// TIA Portal project "Project-Sticle" (V15.1)

(* hardware
DEVICE "S71500/ET200MP station_1"  S7-1500 station
   slot 0: "Rail_0"  Rack  6ES7 590-1***0-0AA0
   slot 1: "PLC_1"  CPU 1513-1 PN  6ES7 513-1AL02-0AB0  V2.6
      slot 3: "CPU display_1"  6ES7591-1AA00-0AA0
*)

// ===== PLC "PLC_1"  CPU 1513-1 PN =====

VAR_GLOBAL   // PLC tag table "Default tag table"
   "Clock_Byte" AT %MB0 : Byte;
   "Clock_10Hz" AT %M0.0 : Bool;
   "Clock_5Hz" AT %M0.1 : Bool;
   "Clock_2.5Hz" AT %M0.2 : Bool;
   "Clock_2Hz" AT %M0.3 : Bool;
   "Clock_1.25Hz" AT %M0.4 : Bool;
   "Clock_1Hz" AT %M0.5 : Bool;
   "Clock_0.625Hz" AT %M0.6 : Bool;
   "Clock_0.5Hz" AT %M0.7 : Bool;
END_VAR

DATA_BLOCK "Avarii"   // DB1
{ S7_Optimized_Access := 'TRUE' }
VERSION : 0.1
   VAR
      esd : Bool;
      esd_btn : Bool;
      reset_esd : Bool;
      confirmare_neprimita_actuator : Bool;
      reset_avarii : Bool;
      avarie_imbuteliere : Bool;
      avarie_capace : Bool;
      avarie_eticheta : Bool;
      avarie_impachetare : Bool;
      avarie_generala : Bool;
   END_VAR
BEGIN
END_DATA_BLOCK

DATA_BLOCK "Alarme"   // DB2
{ S7_Optimized_Access := 'TRUE' }
VERSION : 0.1
   VAR
      alarme_gather : Word;
      alarme_vect : Array[0..15] of Bool;
   END_VAR
BEGIN
END_DATA_BLOCK

DATA_BLOCK "Senzori"   // DB3
{ S7_Optimized_Access := 'TRUE' }
VERSION : 0.1
   VAR
      completat_1 : UInt;
   END_VAR
BEGIN
END_DATA_BLOCK

DATA_BLOCK "Banda"   // DB4
{ S7_Optimized_Access := 'TRUE' }
VERSION : 0.1
   VAR
      banda_pornita_1 : Bool;
      prm_pornire_banda11 : Bool;
      prm_pornire_banda12 : Bool;
      banda_oprita_2 : Bool;
      banda_oprita_3 : Bool;
      banda_oprita_4 : Bool;
   END_VAR
BEGIN
END_DATA_BLOCK

DATA_BLOCK "Aparate"   // DB5
{ S7_Optimized_Access := 'TRUE' }
VERSION : 0.1
   VAR
      numar_sticle_cerut : UInt;
      numar_sticle : UInt;
      inchidere_actuator : Bool;
      deschidere_actuator : Bool;
      confirmare_actuator : Bool;
      timp_umplere_user : Time;
      timp_umplere_secunde : Time;
      terminat_imbuteliere : Bool;
      ajuns_capace : Bool;
      plecat_capace : Bool;
      ajuns_eticheta : Bool;
      plecat_ethicheta : Bool;
      ajuns_impachetare : Bool;
      plecat_impachetare : Bool;
   END_VAR
BEGIN
END_DATA_BLOCK

DATA_BLOCK "Butoane/Permisiuni"   // DB6
{ S7_Optimized_Access := 'TRUE' }
VERSION : 0.1
   VAR
      btn_start : Bool;
      permisiune_start : Bool;
      nr_sticle_complet : Bool;
   END_VAR
BEGIN
END_DATA_BLOCK

DATA_BLOCK "Rising_edges"   // DB7
{ S7_Optimized_Access := 'TRUE' }
VERSION : 0.1
   VAR
      re1 : Bool;
      re2 : Bool;
      re3 : Bool;
   END_VAR
BEGIN
END_DATA_BLOCK

DATA_BLOCK "Hysteresis_DB"   // DB15
{ S7_Optimized_Access := 'TRUE' }
VERSION : 0.1
// stored: InstanceOfName Hysteresis
"Hysteresis"
BEGIN
END_DATA_BLOCK

DATA_BLOCK "Variabile_Hysteresis"   // DB16
{ S7_Optimized_Access := 'TRUE' }
VERSION : 0.1
   VAR
      bool_cond : Bool;
      Hy_val : Real;
      Setpoint : Real;
      temp : Real;
      lim_inf : Real;
      lim_sup : Real;
   END_VAR
BEGIN
END_DATA_BLOCK

// folder: System blocks/Program resources

DATA_BLOCK "timer_confirmare_actuator"   // DB8
{ S7_Optimized_Access := 'TRUE' }
AUTHOR : Simatic
FAMILY : IEC
NAME : IEC_TMR
VERSION : 1.0
// stored: InstanceOfName IEC_TIMER
"IEC_TIMER"
BEGIN
END_DATA_BLOCK

DATA_BLOCK "timer_imbuteliere"   // DB9
{ S7_Optimized_Access := 'TRUE' }
AUTHOR : Simatic
FAMILY : IEC
NAME : IEC_TMR
VERSION : 1.0
// stored: InstanceOfName IEC_TIMER
"IEC_TIMER"
BEGIN
END_DATA_BLOCK

DATA_BLOCK "timer_reset_btn_avarii"   // DB10
{ S7_Optimized_Access := 'TRUE' }
AUTHOR : Simatic
FAMILY : IEC
NAME : IEC_TMR
VERSION : 1.0
// stored: InstanceOfName IEC_TIMER
"IEC_TIMER"
BEGIN
END_DATA_BLOCK

DATA_BLOCK "timer_capace"   // DB11
{ S7_Optimized_Access := 'TRUE' }
AUTHOR : Simatic
FAMILY : IEC
NAME : IEC_TMR
VERSION : 1.0
// stored: InstanceOfName IEC_TIMER
"IEC_TIMER"
BEGIN
END_DATA_BLOCK

DATA_BLOCK "timer_eticheta"   // DB12
{ S7_Optimized_Access := 'TRUE' }
AUTHOR : Simatic
FAMILY : IEC
NAME : IEC_TMR
VERSION : 1.0
// stored: InstanceOfName IEC_TIMER
"IEC_TIMER"
BEGIN
END_DATA_BLOCK

DATA_BLOCK "timer_impachetare"   // DB13
{ S7_Optimized_Access := 'TRUE' }
AUTHOR : Simatic
FAMILY : IEC
NAME : IEC_TMR
VERSION : 1.0
// stored: InstanceOfName IEC_TIMER
"IEC_TIMER"
BEGIN
END_DATA_BLOCK

DATA_BLOCK "reset_esd"   // DB14
{ S7_Optimized_Access := 'TRUE' }
AUTHOR : Simatic
FAMILY : IEC
NAME : IEC_TMR
VERSION : 1.0
// stored: InstanceOfName IEC_TIMER
"IEC_TIMER"
BEGIN
END_DATA_BLOCK

// folder: (top level)

FUNCTION_BLOCK "Hysteresis"   // FB1, LAD
{ S7_Optimized_Access := 'TRUE' }
VERSION : 0.1
   VAR_INPUT
      HY_val : Real;
      Setpoint : Real;
   END_VAR
   VAR_OUTPUT
      h_lim_sup : Real;
      h_lim_inf : Real;
      bool_cond : Bool;
   END_VAR
   VAR_IN_OUT
      temp : Real;
   END_VAR
   VAR
      re1 : Bool;
      re2 : Bool;
      urcare : Bool;
   END_VAR
   VAR_TEMP   // added for the SCL form of the ladder/FBD networks
      _w1 : Bool;
   END_VAR
BEGIN

REGION Network 1: daca are comanda de bool, sa creasca
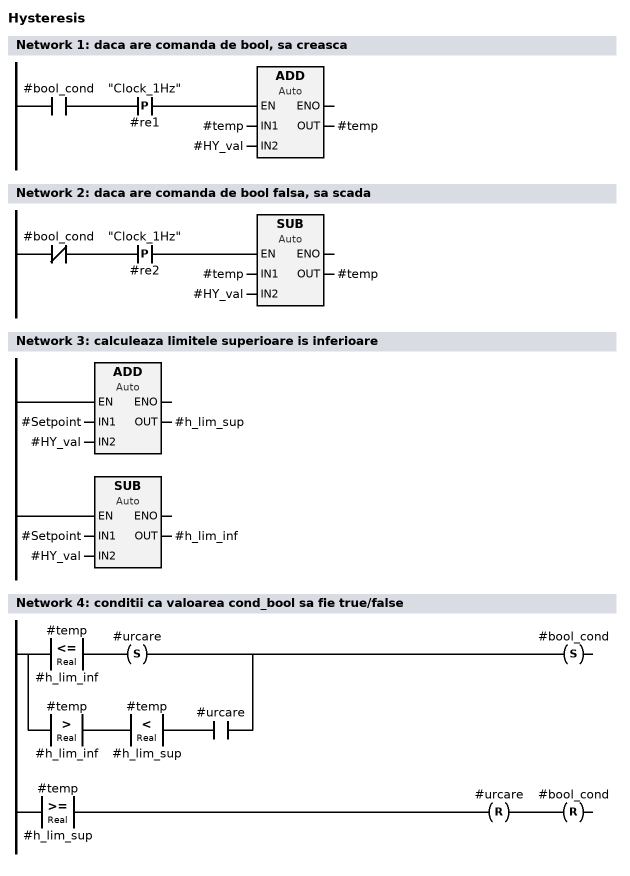
   RUNG wire#powerrail
      Contact( #bool_cond )
      P_Contact(operand := "Clock_1Hz", bit := #re1)
      Add(in1 := #temp, in2 := #HY_val, out => #temp)
   END_RUNG
   // the same network as SCL:
   #_w1 := #bool_cond AND "Clock_1Hz" AND NOT #re1;   // rising edge of "Clock_1Hz"
   #re1 := "Clock_1Hz";
   IF #_w1 THEN #temp := #temp + #HY_val; END_IF;
END_REGION

REGION Network 2: daca are comanda de bool falsa, sa scada
   RUNG wire#powerrail
      I_Contact( #bool_cond )
      P_Contact(operand := "Clock_1Hz", bit := #re2)
      Sub(in1 := #temp, in2 := #HY_val, out => #temp)
   END_RUNG
   // the same network as SCL:
   #_w1 := NOT #bool_cond AND "Clock_1Hz" AND NOT #re2;   // rising edge of "Clock_1Hz"
   #re2 := "Clock_1Hz";
   IF #_w1 THEN #temp := #temp - #HY_val; END_IF;
END_REGION

REGION Network 3: calculeaza limitele superioare is inferioare
   RUNG wire#powerrail
      Add(in1 := #Setpoint, in2 := #HY_val, out => #h_lim_sup)
   END_RUNG
   RUNG wire#powerrail
      Sub(in1 := #Setpoint, in2 := #HY_val, out => #h_lim_inf)
   END_RUNG
   // the same network as SCL:
   #h_lim_sup := #Setpoint + #HY_val;
   #h_lim_inf := #Setpoint - #HY_val;
END_REGION

REGION Network 4: conditii ca valoarea cond_bool sa fie true/false
   RUNG wire#powerrail
      { S7_Templates := "SrcType := Real" } LE_Contact(in1 := #temp, in2 := #h_lim_inf)
      S_Coil( #urcare )
      wire#w1
      S_Coil( #bool_cond )
   END_RUNG
   RUNG wire#powerrail
      { S7_Templates := "SrcType := Real" } GT_Contact(in1 := #temp, in2 := #h_lim_inf)
      { S7_Templates := "SrcType := Real" } LT_Contact(in1 := #temp, in2 := #h_lim_sup)
      Contact( #urcare )
   END_RUNG wire#w1
   RUNG wire#powerrail
      { S7_Templates := "SrcType := Real" } GE_Contact(in1 := #temp, in2 := #h_lim_sup)
      R_Coil( #urcare )
      R_Coil( #bool_cond )
   END_RUNG
   // the same network as SCL:
   #_w1 := #temp <= #h_lim_inf;
   IF #_w1 THEN #urcare := TRUE; END_IF;
   IF #_w1 OR ((#temp > #h_lim_inf) AND (#temp < #h_lim_sup) AND #urcare) THEN #bool_cond := TRUE; END_IF;
   IF #temp >= #h_lim_sup THEN
       #urcare := FALSE;
       #bool_cond := FALSE;
   END_IF;
END_REGION
END_FUNCTION_BLOCK

ORGANIZATION_BLOCK "Main"   // OB1, LAD, ProgramCycle
TITLE = "Main Program Sweep (Cycle)"
{ S7_Optimized_Access := 'TRUE' }
VERSION : 0.1
   VAR_INPUT
      Initial_Call : Bool;   // Initial call of this OB
      Remanence : Bool;   // =True, if remanent data are available
   END_VAR
   VAR_TEMP   // added for the SCL form of the ladder/FBD networks
      _w1 : Bool;
   END_VAR
BEGIN

REGION Network 1: permisiune start(adauga la final si avarie generala pt fiecare aparat in parte)
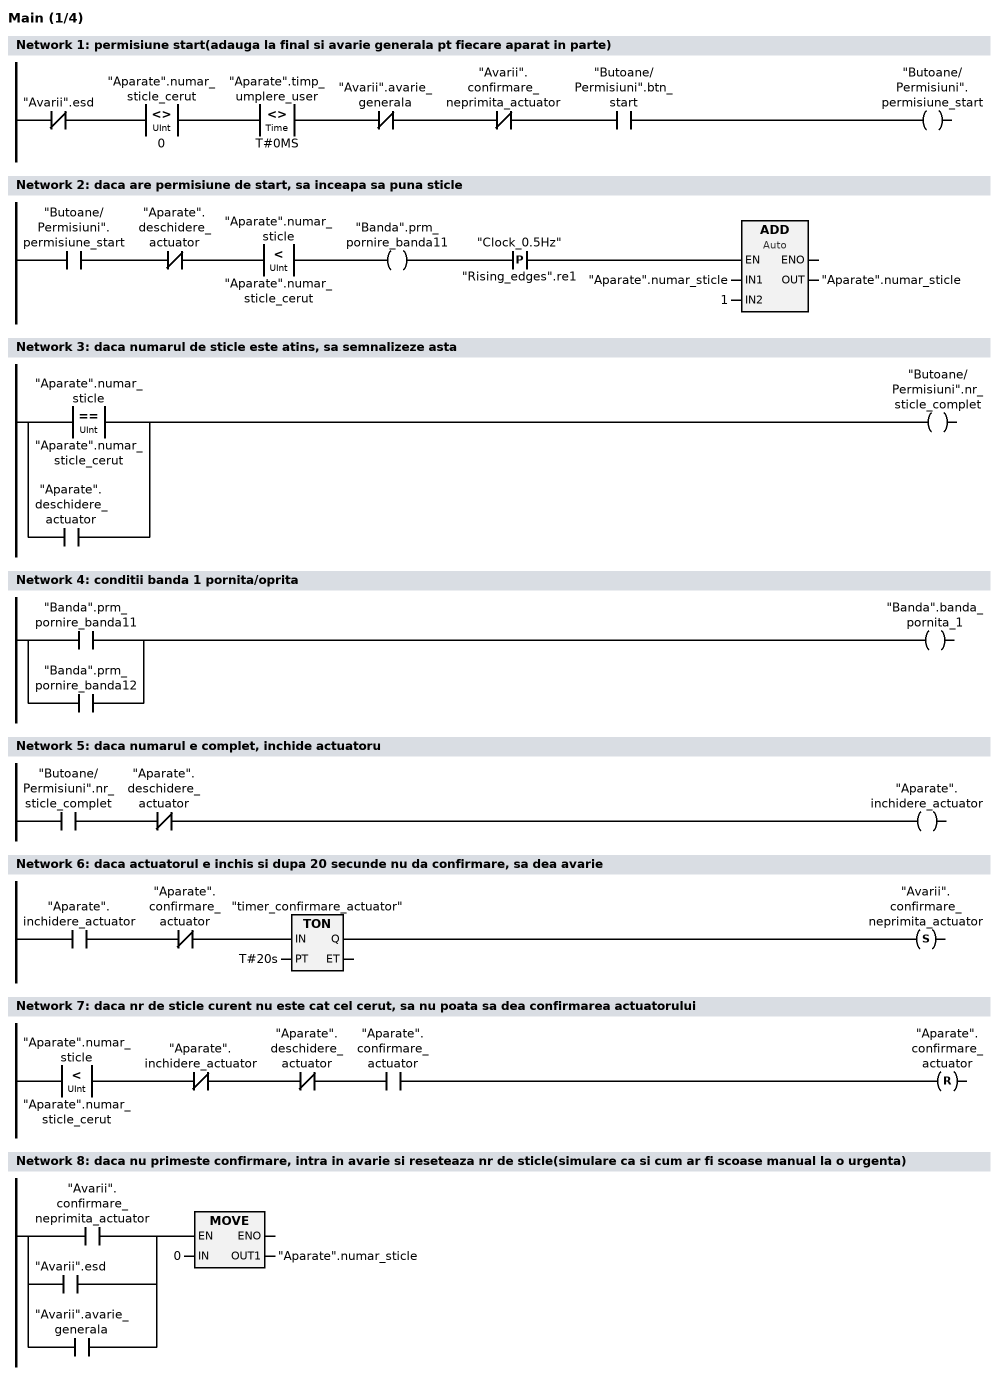
   RUNG wire#powerrail
      I_Contact( "Avarii".esd )
      { S7_Templates := "SrcType := UInt" } NE_Contact(in1 := "Aparate".numar_sticle_cerut, in2 := 0)
      { S7_Templates := "SrcType := Time" } NE_Contact(in1 := "Aparate".timp_umplere_user, in2 := T#0MS)
      I_Contact( "Avarii".avarie_generala )
      I_Contact( "Avarii".confirmare_neprimita_actuator )
      Contact( "Butoane/Permisiuni".btn_start )
      Coil( "Butoane/Permisiuni".permisiune_start )
   END_RUNG
   // the same network as SCL:
   "Butoane/Permisiuni".permisiune_start := NOT "Avarii".esd AND ("Aparate".numar_sticle_cerut <> 0) AND ("Aparate".timp_umplere_user <> T#0MS) AND NOT "Avarii".avarie_generala AND NOT "Avarii".confirmare_neprimita_actuator AND "Butoane/Permisiuni".btn_start;
END_REGION

REGION Network 2: daca are permisiune de start, sa inceapa sa puna sticle
   RUNG wire#powerrail
      Contact( "Butoane/Permisiuni".permisiune_start )
      I_Contact( "Aparate".deschidere_actuator )
      { S7_Templates := "SrcType := UInt" } LT_Contact(in1 := "Aparate".numar_sticle, in2 := "Aparate".numar_sticle_cerut)
      Coil( "Banda".prm_pornire_banda11 )
      P_Contact(operand := "Clock_0.5Hz", bit := "Rising_edges".re1)
      Add(in1 := "Aparate".numar_sticle, in2 := 1, out => "Aparate".numar_sticle)
   END_RUNG
   // the same network as SCL:
   "Banda".prm_pornire_banda11 := "Butoane/Permisiuni".permisiune_start AND NOT "Aparate".deschidere_actuator AND ("Aparate".numar_sticle < "Aparate".numar_sticle_cerut);
   #_w1 := "Banda".prm_pornire_banda11 AND "Clock_0.5Hz" AND NOT "Rising_edges".re1;   // rising edge of "Clock_0.5Hz"
   "Rising_edges".re1 := "Clock_0.5Hz";
   IF #_w1 THEN "Aparate".numar_sticle := "Aparate".numar_sticle + 1; END_IF;
END_REGION

REGION Network 3: daca numarul de sticle este atins, sa semnalizeze asta
   RUNG wire#powerrail
      { S7_Templates := "SrcType := UInt" } EQ_Contact(in1 := "Aparate".numar_sticle, in2 := "Aparate".numar_sticle_cerut)
      wire#w1
      Coil( "Butoane/Permisiuni".nr_sticle_complet )
   END_RUNG
   RUNG wire#powerrail
      Contact( "Aparate".deschidere_actuator )
   END_RUNG wire#w1
   // the same network as SCL:
   "Butoane/Permisiuni".nr_sticle_complet := ("Aparate".numar_sticle = "Aparate".numar_sticle_cerut) OR "Aparate".deschidere_actuator;
END_REGION

REGION Network 4: conditii banda 1 pornita/oprita
   RUNG wire#powerrail
      Contact( "Banda".prm_pornire_banda11 )
      wire#w1
      Coil( "Banda".banda_pornita_1 )
   END_RUNG
   RUNG wire#powerrail
      Contact( "Banda".prm_pornire_banda12 )
   END_RUNG wire#w1
   // the same network as SCL:
   "Banda".banda_pornita_1 := "Banda".prm_pornire_banda11 OR "Banda".prm_pornire_banda12;
END_REGION

REGION Network 5: daca numarul e complet, inchide actuatoru
   RUNG wire#powerrail
      Contact( "Butoane/Permisiuni".nr_sticle_complet )
      I_Contact( "Aparate".deschidere_actuator )
      Coil( "Aparate".inchidere_actuator )
   END_RUNG
   // the same network as SCL:
   "Aparate".inchidere_actuator := "Butoane/Permisiuni".nr_sticle_complet AND NOT "Aparate".deschidere_actuator;
END_REGION

REGION Network 6: daca actuatorul e inchis si dupa 20 secunde nu da confirmare, sa dea avarie
   "timer_confirmare_actuator".TON(IN := "Aparate".inchidere_actuator AND NOT "Aparate".confirmare_actuator,
                           PT := T#20s);
   IF "timer_confirmare_actuator".Q THEN "Avarii".confirmare_neprimita_actuator := TRUE; END_IF;
END_REGION

REGION Network 7: daca nr de sticle curent nu este cat cel cerut, sa nu poata sa dea confirmarea actuatorului
   RUNG wire#powerrail
      { S7_Templates := "SrcType := UInt" } LT_Contact(in1 := "Aparate".numar_sticle, in2 := "Aparate".numar_sticle_cerut)
      I_Contact( "Aparate".inchidere_actuator )
      I_Contact( "Aparate".deschidere_actuator )
      Contact( "Aparate".confirmare_actuator )
      R_Coil( "Aparate".confirmare_actuator )
   END_RUNG
   // the same network as SCL:
   IF ("Aparate".numar_sticle < "Aparate".numar_sticle_cerut) AND NOT "Aparate".inchidere_actuator AND NOT "Aparate".deschidere_actuator AND "Aparate".confirmare_actuator THEN
       "Aparate".confirmare_actuator := FALSE;
   END_IF;
END_REGION

REGION Network 8: daca nu primeste confirmare, intra in avarie si reseteaza nr de sticle(simulare ca si cum ar fi scoase manual la o urgenta)
   RUNG wire#powerrail
      Contact( "Avarii".confirmare_neprimita_actuator )
      wire#w1
      Move(in := 0, out1 => "Aparate".numar_sticle)
   END_RUNG
   RUNG wire#powerrail
      Contact( "Avarii".esd )
   END_RUNG wire#w1
   RUNG wire#powerrail
      Contact( "Avarii".avarie_generala )
   END_RUNG wire#w1
   // the same network as SCL:
   IF "Avarii".confirmare_neprimita_actuator OR "Avarii".esd OR "Avarii".avarie_generala THEN
       "Aparate".numar_sticle := 0;
   END_IF;
END_REGION

REGION Network 9: timp in secunde de la user pt umplere
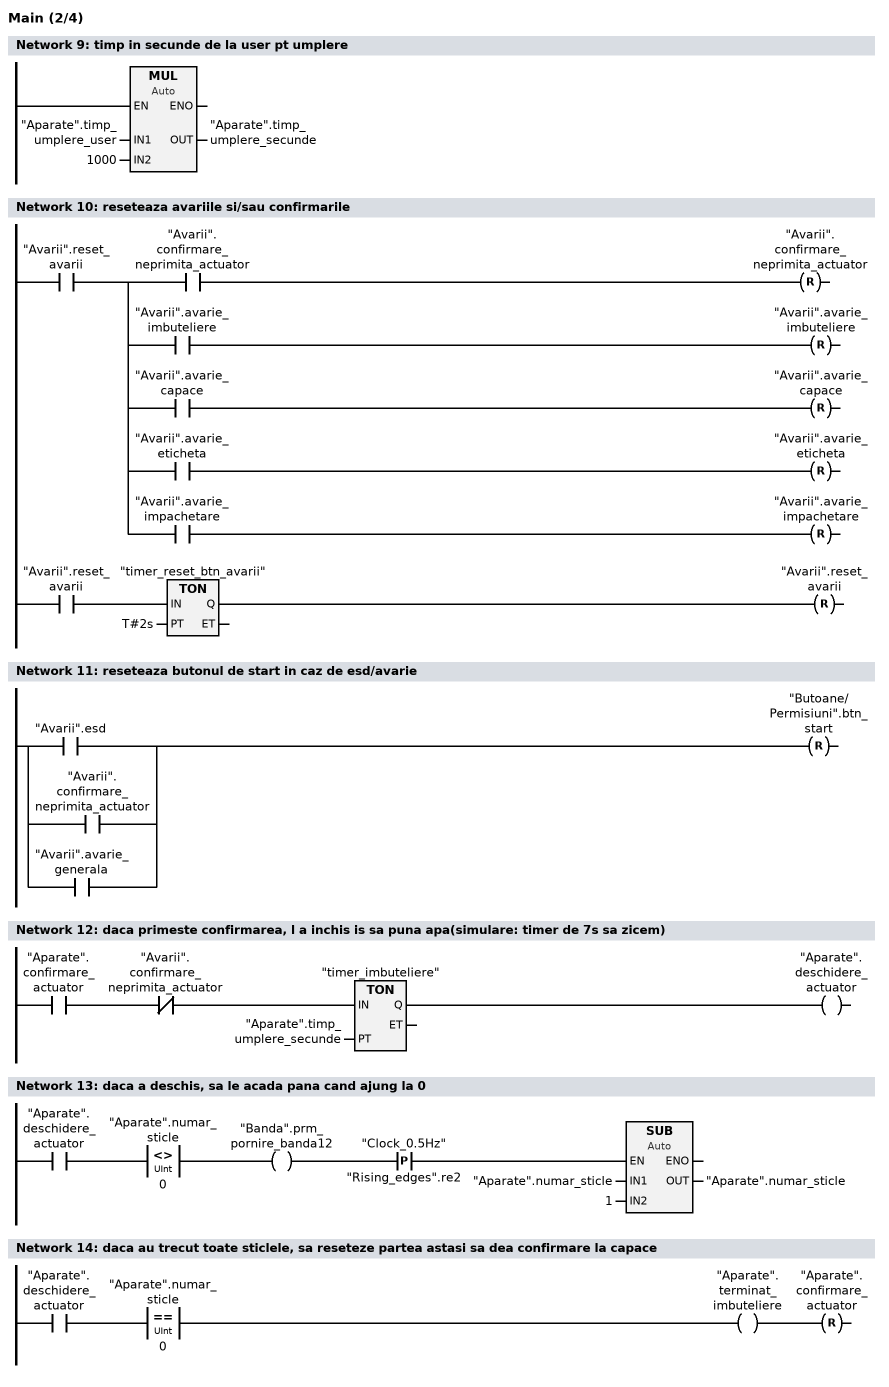
   RUNG wire#powerrail
      Mul(in1 := "Aparate".timp_umplere_user, in2 := 1000, out => "Aparate".timp_umplere_secunde)
   END_RUNG
   // the same network as SCL:
   "Aparate".timp_umplere_secunde := "Aparate".timp_umplere_user * 1000;
END_REGION

REGION Network 10: reseteaza avariile si/sau confirmarile
   IF "Avarii".reset_avarii AND "Avarii".confirmare_neprimita_actuator THEN
       "Avarii".confirmare_neprimita_actuator := FALSE;
   END_IF;
   IF "Avarii".reset_avarii AND "Avarii".avarie_imbuteliere THEN
       "Avarii".avarie_imbuteliere := FALSE;
   END_IF;
   IF "Avarii".reset_avarii AND "Avarii".avarie_capace THEN "Avarii".avarie_capace := FALSE; END_IF;
   IF "Avarii".reset_avarii AND "Avarii".avarie_eticheta THEN "Avarii".avarie_eticheta := FALSE; END_IF;
   IF "Avarii".reset_avarii AND "Avarii".avarie_impachetare THEN
       "Avarii".avarie_impachetare := FALSE;
   END_IF;
   "timer_reset_btn_avarii".TON(IN := "Avarii".reset_avarii, PT := T#2s);
   IF "timer_reset_btn_avarii".Q THEN "Avarii".reset_avarii := FALSE; END_IF;
END_REGION

REGION Network 11: reseteaza butonul de start in caz de esd/avarie
   RUNG wire#powerrail
      Contact( "Avarii".esd )
      wire#w1
      R_Coil( "Butoane/Permisiuni".btn_start )
   END_RUNG
   RUNG wire#powerrail
      Contact( "Avarii".confirmare_neprimita_actuator )
   END_RUNG wire#w1
   RUNG wire#powerrail
      Contact( "Avarii".avarie_generala )
   END_RUNG wire#w1
   // the same network as SCL:
   IF "Avarii".esd OR "Avarii".confirmare_neprimita_actuator OR "Avarii".avarie_generala THEN
       "Butoane/Permisiuni".btn_start := FALSE;
   END_IF;
END_REGION

REGION Network 12: daca primeste confirmarea, l a inchis is sa puna apa(simulare: timer de 7s sa zicem)
   "timer_imbuteliere".TON(IN := "Aparate".confirmare_actuator AND NOT "Avarii".confirmare_neprimita_actuator,
                           PT := "Aparate".timp_umplere_secunde);
   "Aparate".deschidere_actuator := "timer_imbuteliere".Q;
END_REGION

REGION Network 13: daca a deschis, sa le acada pana cand ajung la 0
   RUNG wire#powerrail
      Contact( "Aparate".deschidere_actuator )
      { S7_Templates := "SrcType := UInt" } NE_Contact(in1 := "Aparate".numar_sticle, in2 := 0)
      Coil( "Banda".prm_pornire_banda12 )
      P_Contact(operand := "Clock_0.5Hz", bit := "Rising_edges".re2)
      Sub(in1 := "Aparate".numar_sticle, in2 := 1, out => "Aparate".numar_sticle)
   END_RUNG
   // the same network as SCL:
   "Banda".prm_pornire_banda12 := "Aparate".deschidere_actuator AND ("Aparate".numar_sticle <> 0);
   #_w1 := "Banda".prm_pornire_banda12 AND "Clock_0.5Hz" AND NOT "Rising_edges".re2;   // rising edge of "Clock_0.5Hz"
   "Rising_edges".re2 := "Clock_0.5Hz";
   IF #_w1 THEN "Aparate".numar_sticle := "Aparate".numar_sticle - 1; END_IF;
END_REGION

REGION Network 14: daca au trecut toate sticlele, sa reseteze partea astasi sa dea confirmare la capace
   RUNG wire#powerrail
      Contact( "Aparate".deschidere_actuator )
      { S7_Templates := "SrcType := UInt" } EQ_Contact(in1 := "Aparate".numar_sticle, in2 := 0)
      Coil( "Aparate".terminat_imbuteliere )
      R_Coil( "Aparate".confirmare_actuator )
   END_RUNG
   // the same network as SCL:
   "Aparate".terminat_imbuteliere := "Aparate".deschidere_actuator AND ("Aparate".numar_sticle = 0);
   IF "Aparate".terminat_imbuteliere THEN "Aparate".confirmare_actuator := FALSE; END_IF;
END_REGION

REGION Network 15: daca a terminat imbutelierea, sa seteze ca a ajuns la capace
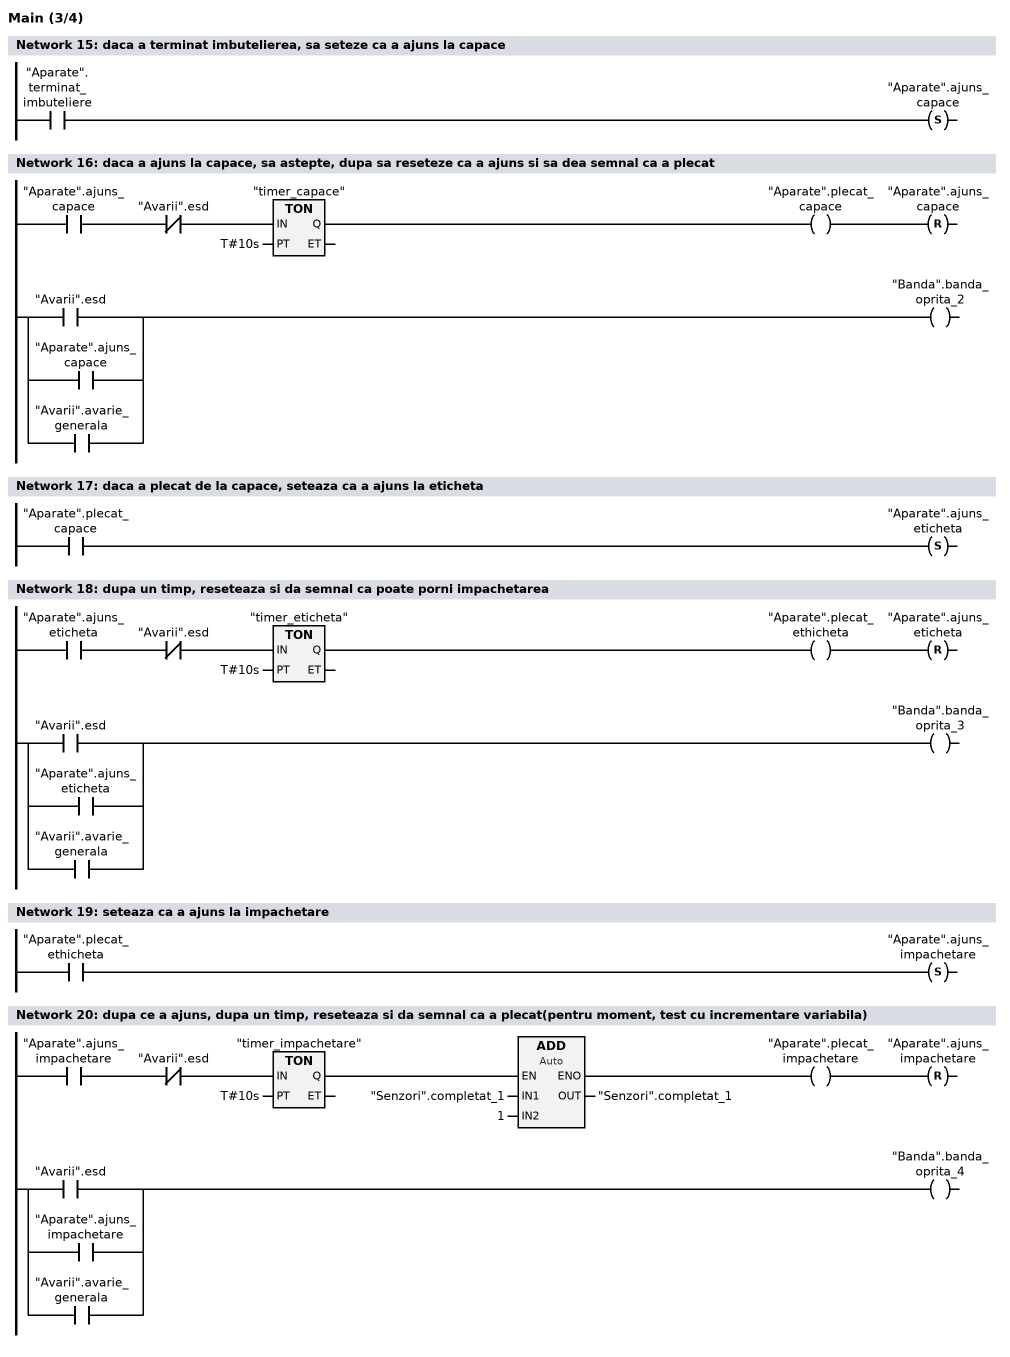
   RUNG wire#powerrail
      Contact( "Aparate".terminat_imbuteliere )
      S_Coil( "Aparate".ajuns_capace )
   END_RUNG
   // the same network as SCL:
   IF "Aparate".terminat_imbuteliere THEN "Aparate".ajuns_capace := TRUE; END_IF;
END_REGION

REGION Network 16: daca a ajuns la capace, sa astepte, dupa sa reseteze ca a ajuns si sa dea semnal ca a plecat
   "timer_capace".TON(IN := "Aparate".ajuns_capace AND NOT "Avarii".esd, PT := T#10s);
   "Aparate".plecat_capace := "timer_capace".Q;
   IF "timer_capace".Q THEN "Aparate".ajuns_capace := FALSE; END_IF;
   "Banda".banda_oprita_2 := "Avarii".esd OR "Aparate".ajuns_capace OR "Avarii".avarie_generala;
END_REGION

REGION Network 17: daca a plecat de la capace, seteaza ca a ajuns la eticheta
   RUNG wire#powerrail
      Contact( "Aparate".plecat_capace )
      S_Coil( "Aparate".ajuns_eticheta )
   END_RUNG
   // the same network as SCL:
   IF "Aparate".plecat_capace THEN "Aparate".ajuns_eticheta := TRUE; END_IF;
END_REGION

REGION Network 18: dupa un timp, reseteaza si da semnal ca poate porni impachetarea
   "timer_eticheta".TON(IN := "Aparate".ajuns_eticheta AND NOT "Avarii".esd, PT := T#10s);
   "Aparate".plecat_ethicheta := "timer_eticheta".Q;
   IF "timer_eticheta".Q THEN "Aparate".ajuns_eticheta := FALSE; END_IF;
   "Banda".banda_oprita_3 := "Avarii".esd OR "Aparate".ajuns_eticheta OR "Avarii".avarie_generala;
END_REGION

REGION Network 19: seteaza ca a ajuns la impachetare
   RUNG wire#powerrail
      Contact( "Aparate".plecat_ethicheta )
      S_Coil( "Aparate".ajuns_impachetare )
   END_RUNG
   // the same network as SCL:
   IF "Aparate".plecat_ethicheta THEN "Aparate".ajuns_impachetare := TRUE; END_IF;
END_REGION

REGION Network 20: dupa ce a ajuns, dupa un timp, reseteaza si da semnal ca a plecat(pentru moment, test cu incrementare variabila)
   "timer_impachetare".TON(IN := "Aparate".ajuns_impachetare AND NOT "Avarii".esd, PT := T#10s);
   IF "timer_impachetare".Q THEN "Senzori".completat_1 := "Senzori".completat_1 + 1; END_IF;
   "Aparate".plecat_impachetare := "timer_impachetare".Q;
   IF "timer_impachetare".Q THEN "Aparate".ajuns_impachetare := FALSE; END_IF;
   "Banda".banda_oprita_4 := "Avarii".esd OR "Aparate".ajuns_impachetare OR "Avarii".avarie_generala;
END_REGION

REGION Network 21: esd btn
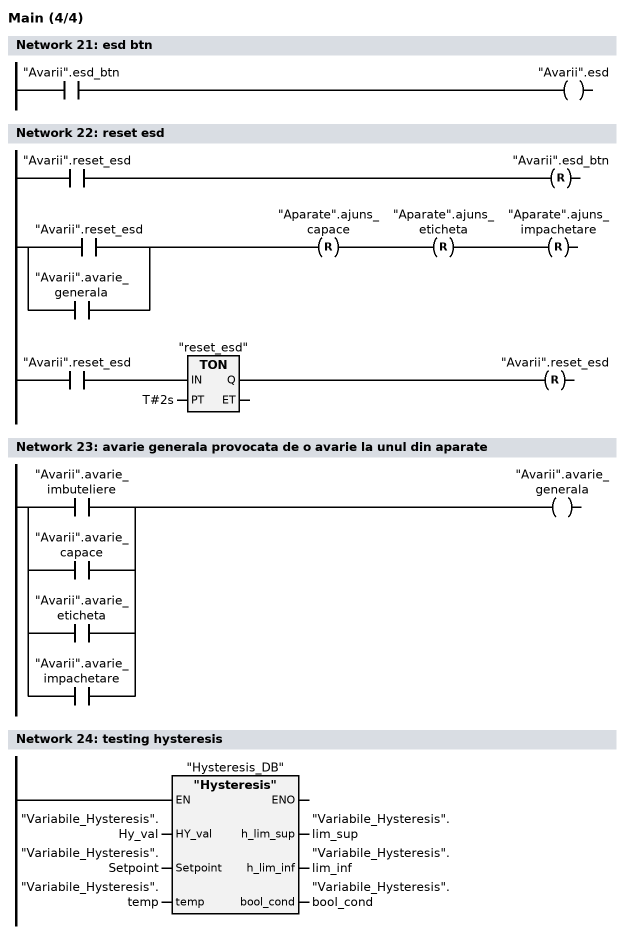
   RUNG wire#powerrail
      Contact( "Avarii".esd_btn )
      Coil( "Avarii".esd )
   END_RUNG
   // the same network as SCL:
   "Avarii".esd := "Avarii".esd_btn;
END_REGION

REGION Network 22: reset esd
   IF "Avarii".reset_esd THEN "Avarii".esd_btn := FALSE; END_IF;
   IF "Avarii".reset_esd OR "Avarii".avarie_generala THEN
       "Aparate".ajuns_capace := FALSE;
       "Aparate".ajuns_eticheta := FALSE;
       "Aparate".ajuns_impachetare := FALSE;
   END_IF;
   "reset_esd".TON(IN := "Avarii".reset_esd, PT := T#2s);
   IF "reset_esd".Q THEN "Avarii".reset_esd := FALSE; END_IF;
END_REGION

REGION Network 23: avarie generala provocata de o avarie la unul din aparate
   RUNG wire#powerrail
      Contact( "Avarii".avarie_imbuteliere )
      wire#w1
      Coil( "Avarii".avarie_generala )
   END_RUNG
   RUNG wire#powerrail
      Contact( "Avarii".avarie_capace )
   END_RUNG wire#w1
   RUNG wire#powerrail
      Contact( "Avarii".avarie_eticheta )
   END_RUNG wire#w1
   RUNG wire#powerrail
      Contact( "Avarii".avarie_impachetare )
   END_RUNG wire#w1
   // the same network as SCL:
   "Avarii".avarie_generala := "Avarii".avarie_imbuteliere OR "Avarii".avarie_capace OR "Avarii".avarie_eticheta OR "Avarii".avarie_impachetare;
END_REGION

REGION Network 24: testing hysteresis
   RUNG wire#powerrail
      "Hysteresis_DB"(HY_val := "Variabile_Hysteresis".Hy_val, Setpoint := "Variabile_Hysteresis".Setpoint, temp := "Variabile_Hysteresis".temp, h_lim_sup => "Variabile_Hysteresis".lim_sup, h_lim_inf => "Variabile_Hysteresis".lim_inf, bool_cond => "Variabile_Hysteresis".bool_cond)
   END_RUNG
   // the same network as SCL:
   "Hysteresis_DB"(HY_val := "Variabile_Hysteresis".Hy_val,   // "Hysteresis"
                   Setpoint := "Variabile_Hysteresis".Setpoint,
                   temp := "Variabile_Hysteresis".temp,
                   h_lim_sup => "Variabile_Hysteresis".lim_sup,
                   h_lim_inf => "Variabile_Hysteresis".lim_inf,
                   bool_cond => "Variabile_Hysteresis".bool_cond);
END_REGION
END_ORGANIZATION_BLOCK